// TIA Portal V20 export
VAR_GLOBAL   // PLC tag table "S2_R1"
   S2_R1_Safety1_1 AT %I550.0 : Bool;
   S2_R1_Safety2_1 AT %I550.1 : Bool;
   S2_R1_Safety3_1 AT %I550.2 : Bool;
   S2_R1_Safety4_1 AT %I550.3 : Bool;
   S2_R1_Safety1_2 AT %I550.4 : Bool;
   S2_R1_Safety2_2 AT %I550.5 : Bool;
   S2_R1_Safety3_2 AT %I550.6 : Bool;
   S2_R1_Safety4_2 AT %I550.7 : Bool;
   S2_R1_Valve_Up AT %Q500.0 : Bool;
   S2_R1_Valve_Down AT %Q500.1 : Bool;
   S2_R1_Sen_Drv_1 AT %I500.0 : Bool;
   S2_R1_Sen_Drv_2 AT %I500.1 : Bool;
   S2_R1_Sen_Drv_3 AT %I500.2 : Bool;
   S2_R1_Sen_Drv_4 AT %I500.3 : Bool;
   S2_R1_Sen_Val1_Up AT %I500.4 : Bool;
   S2_R1_Sen_Val1_Down AT %I500.5 : Bool;
   S2_R1_Sen_Val2_Up AT %I500.6 : Bool;
   S2_R1_Sen_Val2_Down AT %I500.7 : Bool;
   S2_R1_Hyd_Filtr AT %I501.0 : Bool;
   S2_R1_Hyd_Empty AT %I501.1 : Bool;
   SS2_R1_ACK_STO AT %Q150.7 : Bool;
   S2_R1_Hydraulic_Unit AT %Q500.2 : Bool;
END_VAR
